PROGRAM B_2_1_PRG_Master_Station_2

VAR
	eState								: E_Station2_State;
	tonErrorReset						: TON;
	tonStationStopped					: TON;
	ctuErrorCounter						: CTU;
	rGoodStatistics						: R_TRIG;
	rBadStatistics						: R_TRIG;
	rEfficency							: STRING(510);
	
	bPersistentError					: bool;
/////////////////////////////////////////////////////////////////////////////////////I O/////////////////////////////////////////////////////////////////////////////////////	
	bStopped							: BOOL;
	bError								: BOOL;
	bReady								: BOOL;
	bDone								: BOOL;
	bPass								: BOOL;
	bFail								: BOOL;

	
END_VAR

VAR_INPUT	
	
	CMD									:ST_StationCMD;	
	
END_VAR

VAR_OUTPUT	
	
	STATUS								:ST_StationStatus;	
	
END_VAR

B_2_2_PRG_Fault_Station_2( aAlarms := stAlarms );
a_ACT_Ctrl_Station_2();
b_ACT_IO();
c_ACT_Statistics_Station_2();

ACTION a_ACT_Ctrl_Station_2:
/////////////////////////////////////////////////////////////////////////////////////UTILITIES/////////////////////////////////////////////////////////////////////////////////////
tonErrorReset( IN := (eState = E_Station2_State.RESET_ERROR), PT := T#500MS);
tonStationStopped( IN := bStopped, PT := T#1S);
ctuErrorCounter( CU := eState = E_Station2_State.RESET_ERROR, RESET := ((ctuErrorCounter.CV = 5) AND eState = E_Station2_State.PERSISTENT_ERROR), PV := 5, Q => bPersistentError);

/////////////////////////////////////////////////////////////////////////////////////CONDITIONS/////////////////////////////////////////////////////////////////////////////////////

IF (CMD.bAbort OR bError) AND ( eState			= E_Station2_State.HOMING OR
								eState			= E_Station2_State.READY OR
								eState			= E_Station2_State.MOVEMENT_A OR
								eState			= E_Station2_State.MOVEMENT_B OR
								eState			= E_Station2_State.MOVEMENT_C OR
								eState			= E_Station2_State.READY  OR
								eState			= E_Station2_State.DONE) THEN
								
	eState						:= E_Station2_State.STOPPING;
	
END_IF

CASE eState OF
	
	E_Station2_State.ABORTED:
								IF CMD.bEnable AND NOT bError THEN
									eState						:= E_Station2_State.HOMING;
								ELSIF bError THEN
									eState						:= E_Station2_State.ERROR;
								END_IF
	
	E_Station2_State.HOMING:
								IF bReady THEN
									eState						:= E_Station2_State.READY;
								END_IF
	E_Station1_State.RESET:
								stCycleDataStation2.bPass	:= FALSE;
								stCycleDataStation2.bFail	:= FALSE;
								
								eState						:= E_Station2_State.READY;
	E_Station2_State.READY:
								IF CMD.bExecute AND stStation2.Mov1 THEN
									eState						:= E_Station2_State.MOVEMENT_A;
								ELSIF CMD.bExecute AND stStation2.Mov2 THEN
									eState						:= E_Station2_State.MOVEMENT_B;
								ELSIF CMD.bExecute AND stStation2.Mov3 THEN
									eState						:= E_Station2_State.MOVEMENT_C;
								END_IF
	
	E_Station2_State.MOVEMENT_A:
								IF bDone AND stStation2.Mov1 THEN
									eState						:= E_Station2_State.DONE;
								END_IF
	
	E_Station2_State.MOVEMENT_B:
								IF bDone AND stStation2.Mov2 THEN
									eState						:= E_Station2_State.DONE;
								END_IF
	E_Station2_State.MOVEMENT_C:
								IF bDone AND stStation2.Mov3 THEN
									eState						:= E_Station2_State.DONE;
								END_IF
	E_Station2_State.DONE:
								IF  CMD.bReady THEN
									eState						:= E_Station2_State.READY;
								END_IF	
	E_Station1_State.RESULTS:
								
								IF bPass THEN
									stCycleDataStation2.bPass	:= TRUE;
								ELSIF bFail THEN
								 	stCycleDataStation2.bFail	:= TRUE;
								END_IF
								
								IF  CMD.bEndCycle THEN
									eState						:= E_Station2_State.RESET;
								END_IF
/////////////////////////////////////////////////////////////////////////////////////RESET CMD/////////////////////////////////////////////////////////////////////////////////////

	E_Station2_State.STOPPING: 
								IF tonStationStopped.Q THEN
									IF bError THEN
										eState						:= E_Station2_State.ERROR;
									ELSE eState						:= E_Station2_State.ABORTED;
									END_IF

								END_IF
	
	E_Station2_State.ERROR:
								IF NOT bError THEN
									eState						:= E_Station2_State.ABORTED;
								ELSE eState						:= E_Station2_State.RESET_ERROR;
								END_IF
	
	E_Station2_State.RESET_ERROR:
								IF tonErrorReset.Q AND NOT bPersistentError THEN
									eState						:= E_Station2_State.ERROR;
								ELSIF bPersistentError THEN
									eState						:= E_Station2_State.PERSISTENT_ERROR;
								END_IF
	
	E_Station2_State.PERSISTENT_ERROR:
								IF CMD.bReset THEN
									eState						:= E_Station2_State.ERROR;
								END_IF
								
								

ELSE eState := E_Station2_State.ABORTED;
	
END_CASE
/////////////////////////////////////////////////////////////////////////////////////STATUS/////////////////////////////////////////////////////////////////////////////////////

Status.bBusy				:= 	eState			= E_Station2_State.HOMING OR
								eState			= E_Station2_State.MOVEMENT_A OR
								eState			= E_Station2_State.MOVEMENT_B OR
								eState			= E_Station2_State.MOVEMENT_C OR
								eState			= E_Station2_State.STOPPING;
								
Status.bDone				:=	eState			= E_Station2_State.DONE;
											
Status.bError				:= 	eState			= (E_Station2_State.ERROR OR  E_Station2_State.RESET_ERROR OR E_Station2_State.PERSISTENT_ERROR);

Status.bReady				:= 	eState			= E_Station2_State.READY;

Status.bStopped				:= 	eState			= E_Station2_State.ABORTED OR
								eState			= E_Station2_State.READY OR
								eState			= E_Station2_State.ERROR OR
								eState			= E_Station2_State.RESET_ERROR;
END_ACTION

ACTION b_ACT_IO:
//bStopped								:=;
//bError								:=;
//bReady								:=;
//bDone
END_ACTION

ACTION c_ACT_Statistics_Station_2:
stStatisticsHMI[2].sName			:= 'Station 2';


rGoodStatistics( CLK := (stCycleDataStation2.bPass AND (eState = E_Station2_State.RESULTS)) OR bStatisticsTest[2]);
rBadStatistics( CLK := (stCycleDataStation2.bFail AND (eState = E_Station2_State.RESULTS)) OR bStatisticsTest[3]);

IF 	rGoodStatistics.Q THEN
	
	stStatisticsHMI[2].nGood		:= stStatisticsHMI[2].nGood + 1;
	stStatisticsHMI[2].nTotalGood	:= stStatisticsHMI[2].nTotalGood + 1;
	
END_IF
								
IF 	rBadStatistics.Q THEN
	
	stStatisticsHMI[2].nBad			:= stStatisticsHMI[2].nBad + 1;
	stStatisticsHMI[2].nTotalBad	:= stStatisticsHMI[2].nTotalBad + 1;
	
END_IF

IF stStatisticsHMI[2].bResetGood THEN
	stStatisticsHMI[2].nGood		:= 0;
END_IF

IF stStatisticsHMI[2].bResetBad THEN
	stStatisticsHMI[2].nBad			:= 0;
END_IF

IF (( stStatisticsHMI[2].nGood + stStatisticsHMI[2].nBad) <> 0) THEN
	
	rEfficency							:= LREAL_TO_FMTSTR(in := (DINT_TO_REAL(stStatisticsHMI[2].nGood) /( DINT_TO_REAL(stStatisticsHMI[2].nGood) + DINT_TO_REAL(stStatisticsHMI[2].nBad))) * 100.0,iPrecision := 2, bRound := TRUE);
	stStatisticsHMI[2].nEfficency		:= CONCAT(STR1 := '%', STR2 := (rEfficency));

ELSE stStatisticsHMI[2].nEfficency		:= CONCAT(STR1 := '%', STR2 := (DINT_TO_STRING(0)));
	
END_IF
END_ACTION

END_PROGRAM

(* stored: Version 1.1.0.1, ProductVersion 3.1.4024.13
   POU B_2_1_PRG_Master_Station_2: Id {a6876b43-7a04-4227-9137-3bf727782da0}, SpecialFunc None
   Action a_ACT_Ctrl_Station_2: Id {c76df57f-a608-46ce-a480-681c36fd146a}
   Action b_ACT_IO: Id {a6b5537d-697f-4c12-88a8-072e754bb70d}
   Action c_ACT_Statistics_Station_2: Id {a944e097-f352-4ee2-9b3c-c47d97294856} *)
